// TIA Portal V17 export
// export: Created 2024-09-02T12:49:57.8176067Z, ExportSetting WithDefaults, DisplayName Totally Integrated Automation Portal, DisplayVersion V17, DisplayName TIA Portal Openness, DisplayVersion V17, DisplayName TIA Portal Version Control Interface, DisplayVersion V17, DisplayName STEP 7 Professional, DisplayVersion V17, DisplayName STEP 7 Safety, DisplayVersion V17, DisplayName WinCC Professional, DisplayVersion V17
FUNCTION "HLP_Button" : Void   // FC30200, LAD
TITLE = HLP Button / HLP Button
{ S7_Optimized_Access := 'TRUE' }
AUTHOR : OlegFuehrus
FAMILY : HLP
NAME : HLP
VERSION : 1.0
// stored: AutoNumber false, IsIECCheckEnabled false, SetENOAutomatically false, UDAEnableTagReadback false
   VAR_INPUT
      i_FR : Bool;   // Funktionsfreigabe / Functional Approve
      i_FM : Bool;   // Rückmeldung / Feedback
      i_RS : Bool;
   END_VAR
   VAR_IN_OUT
      io_Button : Struct   // Button "Reset"
         Gestaltung : Int;   // Button Anzeige Gestaltung / Button Display Design
         aktiv : Bool;   // Button aktiv (gedrückt) / Button active (pressed)
      END_STRUCT;
   END_VAR
   VAR_TEMP   // added for the SCL form of the ladder/FBD networks
      _w1 : Bool;
   END_VAR
BEGIN

REGION Network 1: Button active (pressed) / Button aktiv (gedrückt)
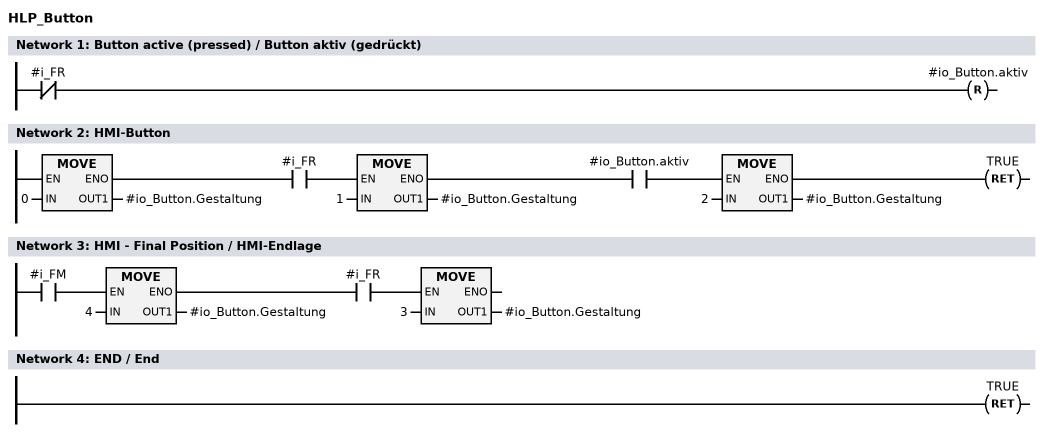
   RUNG wire#powerrail
      I_Contact( #i_FR )
      R_Coil( #io_Button.aktiv )
   END_RUNG
   // the same network as SCL:
   IF NOT #i_FR THEN #io_Button.aktiv := FALSE; END_IF;
END_REGION

REGION Network 2: HMI-Button
   RUNG wire#powerrail
      Move(in := 0, out1 => #io_Button.Gestaltung)
      Contact( #i_FR )
      Move(in := 1, out1 => #io_Button.Gestaltung)
      Contact( #io_Button.aktiv )
      Move(in := 2, out1 => #io_Button.Gestaltung)
      ReturnCoil( TRUE )
   END_RUNG
   // the same network as SCL:
   #io_Button.Gestaltung := 0;
   IF #i_FR THEN #io_Button.Gestaltung := 1; END_IF;
   #_w1 := #i_FR AND #io_Button.aktiv;
   IF #_w1 THEN
       #io_Button.Gestaltung := 2;
       ENO := TRUE;
       RETURN;
   END_IF;
END_REGION

REGION Network 3: HMI - Final Position / HMI-Endlage
   RUNG wire#powerrail
      Contact( #i_FM )
      Move(in := 4, out1 => #io_Button.Gestaltung)
      Contact( #i_FR )
      Move(in := 3, out1 => #io_Button.Gestaltung)
   END_RUNG
   // the same network as SCL:
   IF #i_FM THEN #io_Button.Gestaltung := 4; END_IF;
   IF #i_FM AND #i_FR THEN #io_Button.Gestaltung := 3; END_IF;
END_REGION

REGION Network 4: END / End
   RUNG wire#powerrail
      ReturnCoil( TRUE )
   END_RUNG
   // the same network as SCL:
   ENO := TRUE;
   RETURN;
END_REGION
END_FUNCTION
